(* CODESYS project Box_Sorting.project

Project tree, tasks and I/O mapping:
  Device : CODESYS Control Win V3 x64, 3S - Smart Software Solutions GmbH, version 3.5.16.40
    application Application
      libraries: Standard, * (System)
      task MainTask (cyclic, interval t#20ms, priority 1) calls MainControl
      global variables IOs
      global variables GVL
      Symbols
      visualisation Visualization
      program MainControl [ST]
      program LampCtrl [ST]
      program MainLogic [ST]
      program AlarmHandling [ST]
      program BoxMeasureLogic [ST]
      program SmallBoxLogic [ST]
      program MediumBoxLogic [ST]
      program LargeBoxLogic [ST]
      program AlarmHandlingSUB010 [ST]
      program AlarmHandlingSUB020 [ST]
      program AlarmHandlingSUB030 [ST]
      program AlarmHandlingSUB040 [ST]
      program AlarmHandlingSUB050 [ST]
      program AlarmHandlingCylinder030 [ST]
      program AlarmHandlingCylinder040 [ST]
      program AlarmHandlingCylinder050 [ST]
      program AlarmReset [ST]
  libraries: VisuSymbols, 3.5.10.0 (System)
  text list GlobalTextList
*)

// Device/Application/IOs
VAR_GLOBAL
	//Input
	iSUB010_B1 : BOOL; //Box in position
	iSUB010_B2 : BOOL; //Measure sensor 1, small box
	iSUB010_B3 : BOOL; //Measure sensor 2, medium box
	iSUB010_B4 : BOOL; //Measure sensor 3, large box
	iSUB020_B1 : BOOL; //Small box in position cylinder
	iSUB020_B2 : BOOL; //Medium box in position cylinder
	iSUB020_B3 : BOOL; //Large box in position cylinder
	iSUB030_B1 : BOOL; //Small box first sensor
	iSUB030_B2 : BOOL; //Small box second sensor
	iSUB040_B1 : BOOL; //Medium box first sensor
	iSUB040_B2 : BOOL; //Medium box second sensor
	iSUB050_B1 : BOOL; //Large box first sensor
	iSUB050_B2 : BOOL; //Large box second sensor
	iSUB030_C1_B1 : BOOL; //Small box cylinder max out
	iSUB040_C1_B1 : BOOL; //Medium box cylinder max out
	iSUB050_C1_B1 : BOOL; //Large box cylinder max out
	
	//Output
	oSUB000_H4 : BOOL; //Green light
	oSUB000_H5 : BOOL; //Amber light
	oSUB000_H6 : BOOL; //Red light
	oSUB010_K1 : BOOL; //Sort conveyor
	oSUB020_K1 : BOOL; //Transport conveyor
	oSUB030_K1 : BOOL; //Small box conveyor
	oSUB040_K1 : BOOL; //Medium box conveyor
	oSUB050_K1 : BOOL; //Large box conveyor
	oSUB030_Y1 : BOOL; //Small box cylinder
	oSUB040_Y1 : BOOL; //Medium box cylinder
	oSUB050_Y1 : BOOL; //Large box cylinder

END_VAR

// Device/Application/GVL
VAR_GLOBAL
	
	(*HMI INPUTS*)
	iSUB000_S1: BOOL; 	// Start button
	iSUB000_S2: BOOL := TRUE;  	// Stop button (NC)
	iSUB000_S3: BOOL;	// Reset button

	(*HMI OUTPUTS*)
	oSUB000_H1: BOOL; 	// Start button lamp
	oSUB000_H2: INT; 	// Display
	oSUB000_H3: BOOL; 	// Reset button lamp

END_VAR

// Device/Application/MainControl
PROGRAM MainControl
VAR_INPUT
    iStart : BOOL;   // Start
    iStop  : BOOL;   // Stop
    iFault : BOOL;   // Fault
END_VAR

VAR_OUTPUT
    oRun         : BOOL;   // State Run
    oIdle        : BOOL;   // State Idle
    oFaultActive : BOOL;   // State Faulty
END_VAR

VAR
    Mode : INT := 0;  // 0=Idle, 1=Run, 2=Fault
	prevSUB010_K1 : BOOL;
	prevSUB020_K1 : BOOL;
	prevSUB030_K1 : BOOL;
	prevSUB040_K1 : BOOL;
	prevSUB050_K1 : BOOL;
	valueSaved :BOOL;
	backupSUB010_K1 : BOOL;
	backupSUB020_K1 : BOOL;
	backupSUB030_K1 : BOOL;
	backupSUB040_K1 : BOOL;
	backupSUB050_K1 : BOOL;

	//boxInTransport : BOOL; //a box are deployed and are in transit
END_VAR

AlarmHandling();
iFault := AlarmHandling.alarmActive;

// Huvudlogik
CASE Mode OF
    0: // Idle
        oRun := FALSE;
        oIdle := TRUE;
        oFaultActive := FALSE;
		
		//Save outputs when enter Idle
		IF NOT valueSaved AND NOT iFault THEN
			backupSUB010_K1 := IOs.oSUB010_K1;
			backupSUB020_K1 := IOs.oSUB020_K1;
			backupSUB030_K1 := IOs.oSUB030_K1;
			backupSUB040_K1 := IOs.oSUB040_K1;
			backupSUB050_K1 := IOs.oSUB050_K1;
			valueSaved := TRUE;
		END_IF
        
        IF GVL.iSUB000_S1 THEN //Start
			iStop := FALSE;
			iStart := TRUE;
			IF NOT iFault THEN
            	Mode := 1; // Automatic operation
        	ELSE
            	Mode := 2; //Faulted
			END_IF;
        END_IF;
		
		//Stop output in Idle
		IOs.oSUB010_K1 := FALSE;
		IOs.oSUB020_K1 := FALSE;
		IOs.oSUB030_K1 := FALSE;
		IOs.oSUB040_K1 := FALSE;
		IOs.oSUB050_K1 := FALSE;
		
    1: // Run (Automatic)
        oRun := TRUE;
        oIdle := FALSE;
        oFaultActive := FALSE;
        
		//Restore backup for outputs when we start
		IF valueSaved THEN
			IOs.oSUB010_K1 := backupSUB010_K1;
			IOs.oSUB020_K1 := backupSUB020_K1;
			IOs.oSUB030_K1 := backupSUB030_K1;
			IOs.oSUB040_K1 := backupSUB040_K1;
			IOs.oSUB050_K1 := backupSUB050_K1;
			valueSaved := FALSE;
		END_IF
		
		//Enter Faulty if alarm active
		IF iFault THEN
			//Save all output when alarm
			IF NOT valueSaved THEN
				backupSUB010_K1 := IOs.oSUB010_K1;
				backupSUB020_K1 := IOs.oSUB020_K1;
				backupSUB030_K1 := IOs.oSUB030_K1;
				backupSUB040_K1 := IOs.oSUB040_K1;
				backupSUB050_K1 := IOs.oSUB050_K1;
				valueSaved := TRUE;
			END_IF;
			//Stop output when fault
			IOs.oSUB010_K1 := FALSE;
			IOs.oSUB020_K1 := FALSE;
			IOs.oSUB030_K1 := FALSE;
			IOs.oSUB040_K1 := FALSE;
			IOs.oSUB050_K1 := FALSE;
			
			Mode := 2; //Faulted
		ELSIF NOT GVL.iSUB000_S2 THEN
			iStop := TRUE;
			iStart := FALSE;
			Mode := 0; // Set Idle mode
		ELSE
			MainLogic();
		END_IF
        

    2: // Faulted
        oRun := FALSE;
        oIdle := FALSE;
        oFaultActive := TRUE;
		
		//Stop output when fault
		IOs.oSUB010_K1 := FALSE;
		IOs.oSUB020_K1 := FALSE;
		IOs.oSUB030_K1 := FALSE;
		IOs.oSUB040_K1 := FALSE;
		IOs.oSUB050_K1 := FALSE;
		
		IF GVL.iSUB000_S3 THEN
			iStop := TRUE;
			iStart := FALSE;
			AlarmReset();
			IF NOT IOs.iSUB010_B1 THEN // Prevent alarm 9 to heal if before second box is removed from system
				Mode := 0; // Return to idle
			ELSE //Still keep alarm 9
				AlarmHandling.alarmActive := TRUE;
				AlarmHandling.alarmCode := 9;	
			END_IF
        END_IF;

    ELSE
        Mode := 0; // Failsafe
END_CASE;

//Call lamp control
LampCtrl();

END_PROGRAM

// Device/Application/AlarmHandling
PROGRAM AlarmHandling
VAR_INPUT
	boxInSystem : BOOL; //Box introduced in the system
	alarmActive : BOOL; //If any alarm is active
	alarmCode : INT;  //Alarm code
END_VAR
VAR
END_VAR

//Stop all timers if a alarm is active
IF alarmCode <> 0 THEN
	AlarmHandlingSUB010.startTimeSUB010 := FALSE;
	AlarmHandlingSUB020.startTimeSUB020 := FALSE;
	AlarmHandlingSUB030.startTimeSUB030 := FALSE;
	AlarmHandlingSUB040.startTimeSUB040 := FALSE;
	AlarmHandlingSUB050.startTimeSUB050 := FALSE;
	AlarmHandlingCylinder030.startTimeCyl030 := FALSE;
	AlarmHandlingCylinder040.startTimeCyl040 := FALSE;
	AlarmHandlingCylinder050.startTimeCyl050 := FALSE;
END_IF
AlarmHandlingSUB010();
AlarmHandlingSUB020();
AlarmHandlingSUB030();
AlarmHandlingSUB040();
AlarmHandlingSUB050();
AlarmHandlingCylinder030();
AlarmHandlingCylinder040();
AlarmHandlingCylinder050();

//Display the Alarm code
oSUB000_H2 := alarmCode;

END_PROGRAM

// Device/Application/AlarmHandlingSUB010
PROGRAM AlarmHandlingSUB010
VAR_INPUT
	startTimeSUB010 : BOOL; //Activate timer
	SUB010Timer : TON;  //Alarm timer
END_VAR
VAR
	boxStart : F_TRIG; // Instance of flankdetector, control when box is on the conveyour
END_VAR

//Alarmhandling Conveyour 1, SUB010
boxStart(CLK := IOs.iSUB010_B1);
IF boxStart.Q THEN
	AlarmHandling.boxInSystem := TRUE;
	startTimeSUB010 := TRUE;
ELSIF IOs.iSUB010_B1 AND AlarmHandling.boxInSystem AND NOT MainControl.iStop THEN
	AlarmHandling.alarmActive := TRUE;
	IF AlarmHandling.alarmCode = 0 THEN
		AlarmHandling.alarmCode := 9;
	END_IF;
END_IF
IF IOs.iSUB010_B2 OR MainControl.iStop THEN //Cancel alarm
	startTimeSUB010 := FALSE;
END_IF
IF SUB010Timer.Q AND (AlarmHandling.alarmCode = 0) THEN
	AlarmHandling.alarmActive := TRUE;
	AlarmHandling.alarmCode := 1;
END_IF
SUB010Timer(IN := startTimeSUB010, PT := T#4S);

END_PROGRAM

// Device/Application/AlarmHandlingSUB020
PROGRAM AlarmHandlingSUB020
VAR_INPUT
	startTimeSUB020 : BOOL; //Activate timer
	SUB020Timer : TON;  //Alarm timer
END_VAR
VAR
END_VAR

//Alarmhandling Conveyour 2, SUB020
IF IOs.iSUB010_B2 AND (AlarmHandling.alarmCode = 0) AND NOT MainControl.iStop THEN
	startTimeSUB020 := TRUE;
END_IF
IF IOs.iSUB020_B1 AND (MainLogic.boxSize = 1) THEN //Cancel alarm when reach small box sensor, small box
	startTimeSUB020 := FALSE;
ELSIF IOs.iSUB020_B2 AND (MainLogic.boxSize = 2) THEN //Cancel alarm when reach medium box sensor, medium box
	startTimeSUB020 := FALSE;
ELSIF IOs.iSUB020_B3 AND (MainLogic.boxSize = 3) THEN //Cancel alarm when reach large box sensor, large box
	startTimeSUB020 := FALSE;
ELSIF MainControl.iStop THEN
	startTimeSUB020 := FALSE;
END_IF
IF SUB020Timer.Q AND (AlarmHandling.alarmCode = 0) THEN
	AlarmHandling.alarmActive := TRUE;
	AlarmHandling.alarmCode := 2;
END_IF
SUB020Timer(IN := startTimeSUB020, PT := T#8S);

END_PROGRAM

// Device/Application/MainLogic
PROGRAM MainLogic
VAR_INPUT
	boxSize : INT; //Size of the Box
END_VAR
VAR
END_VAR

IF boxSize = 0 THEN  //Box to measure
	BoxMeasureLogic();
ELSIF boxSize = 1 THEN //Small box
	SmallBoxLogic();
ELSIF BoxSize = 2 THEN //Medium box
	MediumBoxLogic();
ELSIF boxSize = 3 THEN //Large box
	LargeBoxLogic();
END_IF

END_PROGRAM

// Device/Application/BoxMeasureLogic
PROGRAM BoxMeasureLogic
VAR
END_VAR

//Start conveyor 1
IF MainControl.oRun AND IOs.iSUB010_B1 THEN
	IOs.oSUB010_K1 := TRUE;
END_IF
//Measure Box size, Small =1, Medium =2, Large =3.
IF IOs.iSUB010_B2 THEN
	MainLogic.boxSize := 1;
	IF IOs.iSUB010_B3 THEN
		MainLogic.boxSize := 2;
		IF IOs.iSUB010_B4 THEN
			MainLogic.boxSize := 3;
		END_IF
	END_IF
END_IF
//Start conveyor 2
IF MainLogic.boxSize > 0 AND IOs.oSUB010_K1 THEN
	IOs.oSUB020_K1 := TRUE;
END_IF

END_PROGRAM

// Device/Application/SmallBoxLogic
PROGRAM SmallBoxLogic
VAR
END_VAR

//Check if Box size is small at cylinder_small. If small Box, stop conveyor and push Box to conveyor 3
IF IOs.iSUB020_B1 THEN
	IOs.oSUB010_K1 := FALSE; //Stop conveyor 1
	IF MainLogic.boxSize = 1 THEN
		IOs.oSUB020_K1 := FALSE; //Stop conveyor 2
		IOs.oSUB030_Y1 := TRUE;  //Expand cylinder small
	END_IF
END_IF

//When cylinder small is fully out and first sensor on conveyor 3 is akitve, start conveyor 3
IF IOs.iSUB030_C1_B1 AND IOs.iSUB030_B1 THEN
	IOs.oSUB030_Y1 := FALSE;  //Retract cylinder small
	IOs.oSUB030_K1 := TRUE;
END_IF

//Stop conveyor 3 when it reach second sensor
IF IOs.iSUB030_B2 THEN
	IOs.oSUB030_K1 := FALSE;
	MainLogic.boxSize := 0;
END_IF

END_PROGRAM

// Device/Application/MediumBoxLogic
PROGRAM MediumBoxLogic
VAR
END_VAR

//Check if Box size is medium at cylinder_medium. If medium Box, stop conveyor and push Box to conveyor 4
IF MainLogic.boxSize = 2 AND IOs.iSUB020_B2 THEN
	IOs.oSUB010_K1 := FALSE; //Stop conveyor 1
	IOs.oSUB020_K1 := FALSE; //Stop conveyor 2
	IOs.oSUB040_Y1 := TRUE;  //Expand cylinder medium
END_IF

//When cylinder medium is fully out and first sensor on conveyor 4 is akitve, start conveyor 4
IF IOs.iSUB040_C1_B1 AND IOs.iSUB040_B1 THEN
	IOs.oSUB040_Y1 := FALSE;  //Retract cylinder medium
	IOs.oSUB040_K1 := TRUE; //Start conveyor 4
END_IF

//Stop conveyor 4 when it reach second sensor
IF IOs.iSUB040_B2 THEN
	IOs.oSUB040_K1 := FALSE;
	MainLogic.boxSize := 0;
END_IF

END_PROGRAM

// Device/Application/LargeBoxLogic
PROGRAM LargeBoxLogic
VAR
END_VAR

//Check if Box size is large at cylinder_large. If large Box, stop conveyor and push Box to conveyor 5
IF MainLogic.boxSize = 3 AND IOs.iSUB020_B3 THEN
	IOs.oSUB010_K1 := FALSE; //Stop conveyor 1
	IOs.oSUB020_K1 := FALSE; //Stop conveyor 2
	IOs.oSUB050_Y1 := TRUE;  //Expand cylinder large
END_IF

//When cylinder large is fully out and first sensor on conveyor 5 is aktive, start conveyor 5
IF IOs.iSUB050_C1_B1 AND IOs.iSUB050_B1 THEN
	IOs.oSUB050_Y1 := FALSE;  //Retract cylinder large
	IOs.oSUB050_K1 := TRUE; //Start conveyor 5
END_IF

//Stop conveyor 5 when it reach second sensor
IF IOs.iSUB050_B2 THEN
	IOs.oSUB050_K1 := FALSE;
	MainLogic.boxSize := 0;
END_IF

END_PROGRAM

// Device/Application/AlarmHandlingSUB030
PROGRAM AlarmHandlingSUB030
VAR_INPUT
	startTimeSUB030 : BOOL; //Activate timer
	SUB030Timer : TON; //Alarm timer
END_VAR
VAR
	boxEndSmall : F_TRIG; // Instance of flankdetector, control when box is removed
END_VAR

//Alarmhandling Conveyour 3, SUB030
IF IOs.iSUB030_B1 AND (AlarmHandling.alarmCode = 0) AND NOT MainControl.iStop THEN
	startTimeSUB030 := TRUE;
END_IF
boxEndSmall(CLK := IOs.iSUB030_B2);
IF boxEndSmall.Q THEN //Cancel alarm
	startTimeSUB030 := FALSE;
	IF NOT IOs.iSUB030_B2 THEN
		AlarmHandling.boxInSystem := FALSE;
	END_IF
ELSIF MainControl.iStop THEN
	startTimeSUB030 := FALSE;
END_IF
IF SUB030Timer.Q AND (AlarmHandling.alarmCode = 0) THEN
	AlarmHandling.alarmActive := TRUE;
	AlarmHandling.alarmCode := 3;
END_IF
SUB030Timer(IN := startTimeSUB030, PT := T#7.2S);

END_PROGRAM

// Device/Application/AlarmHandlingSUB040
PROGRAM AlarmHandlingSUB040
VAR_INPUT
	startTimeSUB040 : BOOL; //Activate timer
	SUB040Timer : TON;  //Alarm timer
END_VAR
VAR
	boxEndMedium : F_TRIG; // Instance of flankdetector, control when box is removed
END_VAR

//Alarmhandling Conveyour 4, SUB040
IF IOs.iSUB040_B1 AND (AlarmHandling.alarmCode = 0) AND NOT MainControl.iStop THEN
	startTimeSUB040 := TRUE;
END_IF
boxEndMedium(CLK := IOs.iSUB040_B2);
IF boxEndMedium.Q THEN //Cancel alarm
	startTimeSUB040 := FALSE;
	IF NOT IOs.iSUB040_B2 THEN
		AlarmHandling.boxInSystem := FALSE;
	END_IF
ELSIF MainControl.iStop THEN
	startTimeSUB040 := FALSE;
END_IF
IF SUB040Timer.Q AND (AlarmHandling.alarmCode = 0) THEN
	AlarmHandling.alarmActive := TRUE;
	AlarmHandling.alarmCode := 4;
END_IF
SUB040Timer(IN := startTimeSUB040, PT := T#7.3S);

END_PROGRAM

// Device/Application/AlarmHandlingSUB050
PROGRAM AlarmHandlingSUB050
VAR_INPUT
	startTimeSUB050 : BOOL; //Activate timer
	SUB050Timer : TON;  //Alarm timer
END_VAR
VAR
	boxEndLarge : F_TRIG; // Instance of flankdetector, control when box is removed
END_VAR

//Alarmhandling Conveyour 5, SUB050
IF IOs.iSUB050_B1 AND (AlarmHandling.alarmCode = 0) AND NOT MainControl.iStop THEN
	startTimeSUB050 := TRUE;
END_IF
boxEndLarge(CLK := IOs.iSUB050_B2);
IF boxEndLarge.Q THEN //Cancel alarm
	startTimeSUB050 := FALSE;
	IF NOT IOs.iSUB050_B2 THEN
		AlarmHandling.boxInSystem := FALSE;
	END_IF
ELSIF MainControl.iStop THEN
	startTimeSUB050 := FALSE;
END_IF
IF SUB050Timer.Q AND (AlarmHandling.alarmCode = 0) THEN
	AlarmHandling.alarmActive := TRUE;
	AlarmHandling.alarmCode := 5;
END_IF
SUB050Timer(IN := startTimeSUB050, PT := T#7.4S);

END_PROGRAM

// Device/Application/AlarmHandlingCylinder030
PROGRAM AlarmHandlingCylinder030
VAR_INPUT
	Cyl030Timer : TON; //Alarm timer
	startTimeCyl030 : BOOL; //Activate timer
END_VAR
VAR
END_VAR

//Alarmhandling Cylinder small, SUB030Cylinder
//Cylinder do not expand
IF IOs.iSUB020_B1 AND (MainLogic.boxSize = 1) AND NOT MainControl.iStop THEN
	startTimeCyl030 := TRUE;
END_IF
IF IOs.iSUB030_B1 THEN //Cancel alarm
	startTimeCyl030 := FALSE;
END_IF
IF Cyl030Timer.Q AND (AlarmHandling.alarmCode = 0) THEN
	AlarmHandling.alarmActive := TRUE;
	AlarmHandling.alarmCode := 6;
END_IF
Cyl030Timer(IN := startTimeCyl030, PT := T#6.5S);

END_PROGRAM

// Device/Application/AlarmHandlingCylinder040
PROGRAM AlarmHandlingCylinder040
VAR_INPUT
	Cyl040Timer : TON; //Alarm timer
	startTimeCyl040 : BOOL; //Activate timer
END_VAR
VAR
END_VAR

//Alarmhandling Cylinder medium, SUB040Cylinder
//Cylinder do not expand
IF IOs.iSUB020_B2 AND (MainLogic.boxSize = 2) AND NOT MainControl.iStop THEN
	startTimeCyl040 := TRUE;
END_IF
IF IOs.iSUB040_B1 THEN //Cancel alarm
	startTimeCyl040 := FALSE;
END_IF
IF Cyl040Timer.Q AND (AlarmHandling.alarmCode = 0) THEN
	AlarmHandling.alarmActive := TRUE;
	AlarmHandling.alarmCode := 7;
END_IF
Cyl040Timer(IN := startTimeCyl040, PT := T#6.6S);

END_PROGRAM

// Device/Application/AlarmHandlingCylinder050
PROGRAM AlarmHandlingCylinder050
VAR_INPUT
	Cyl050Timer : TON; //Alarm timer
	startTimeCyl050 : BOOL; //Activate timer
END_VAR
VAR
END_VAR

//Alarmhandling Cylinder large, SUB050Cylinder
//Cylinder do not expand
IF IOs.iSUB020_B3 AND (MainLogic.boxSize = 3) AND NOT MainControl.iStop THEN
	startTimeCyl050 := TRUE;
END_IF
IF IOs.iSUB050_B1 THEN //Cancel alarm
	startTimeCyl050 := FALSE;
END_IF
IF Cyl050Timer.Q AND (AlarmHandling.alarmCode = 0) THEN
	AlarmHandling.alarmActive := TRUE;
	AlarmHandling.alarmCode := 8;
END_IF
Cyl050Timer(IN := startTimeCyl050, PT := T#6.7S);

END_PROGRAM

// Device/Application/AlarmReset
PROGRAM AlarmReset
VAR
END_VAR

//Reset alarm
AlarmHandling.alarmActive := FALSE;
AlarmHandlingSUB010.startTimeSUB010 := FALSE;
AlarmHandlingSUB020.startTimeSUB020 := FALSE;
AlarmHandlingSUB030.startTimeSUB030 := FALSE;
AlarmHandlingSUB040.startTimeSUB040 := FALSE;
AlarmHandlingSUB050.startTimeSUB050 := FALSE;
AlarmHandlingSUB010.SUB010Timer(IN := AlarmHandlingSUB010.startTimeSUB010);
AlarmHandlingSUB020.SUB020Timer(IN := AlarmHandlingSUB020.startTimeSUB020);
AlarmHandlingSUB030.SUB030Timer(IN := AlarmHandlingSUB030.startTimeSUB030);
AlarmHandlingSUB040.SUB040Timer(IN := AlarmHandlingSUB040.startTimeSUB040);
AlarmHandlingSUB050.SUB050Timer(IN := AlarmHandlingSUB050.startTimeSUB050);
AlarmHandlingCylinder030.startTimeCyl030 := FALSE;
AlarmHandlingCylinder040.startTimeCyl040 := FALSE;
AlarmHandlingCylinder050.startTimeCyl050 := FALSE;
AlarmHandlingCylinder030.Cyl030Timer(IN := AlarmHandlingCylinder030.startTimeCyl030);
AlarmHandlingCylinder040.Cyl040Timer(IN := AlarmHandlingCylinder040.startTimeCyl040);
AlarmHandlingCylinder050.Cyl050Timer(IN := AlarmHandlingCylinder050.startTimeCyl050);
AlarmHandling.alarmCode := 0;

END_PROGRAM

// Device/Application/LampCtrl
PROGRAM LampCtrl
VAR
	GreenBlink : TON; //Green light blink timer
	RedBlink : TON;   //Red light blink timer 
END_VAR

IF MainControl.oRun THEN
	IOs.oSUB000_H4 := TRUE;
	IOs.oSUB000_H5 := FALSE;
	IOs.oSUB000_H6 := FALSE;
	oSUB000_H1 := TRUE;
	oSUB000_H3 := FALSE;
ELSIF MainControl.oIdle THEN
	IOs.oSUB000_H4 := FALSE;
	IOs.oSUB000_H5 := TRUE;
	IOs.oSUB000_H6 := FALSE;
	GreenBlink(IN := NOT GreenBlink.Q, PT := T#2S);
	oSUB000_H1 := GreenBlink.ET > T#1S; //Green shall blink in IDLE
	oSUB000_H3 := FALSE;
ELSIF MainControl.oFaultActive THEN
	IOs.oSUB000_H4 := FALSE;
	IOs.oSUB000_H5 := FALSE;
	oSUB000_H1 := FALSE;
	RedBlink(IN := NOT RedBlink.Q, PT := T#2S);
	IOs.oSUB000_H6 := oSUB000_H3 := RedBlink.ET > T#1S; //Red shall blink in Faulty
END_IF

END_PROGRAM

// Device/Application/Visualization
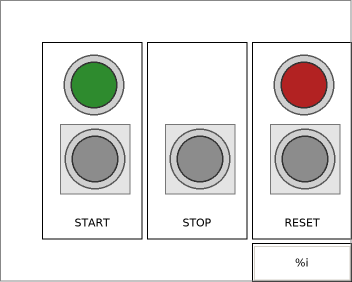
VISUALIZATION Visualization  // 352x282
    Rectangle (42,42 100x197)
    Lamp1 (59,50 70x70), variable: oSUB000_H1, style: Lamp-Lamp1-Green
    PushSwitch (60,124 70x70), variable: iSUB000_S1, behaviour: TAP, style: Switch-PushSwitch-Gray
    Label (46,208 92x30), "START"
    Rectangle (147,42 100x197)
    PushSwitch (165,124 70x70), variable: iSUB000_S2, behaviour: TAP, style: Switch-PushSwitch-Gray
    Label (151,208 92x30), "STOP"
    Rectangle (252,42 100x197)
    Lamp1 (269,50 70x70), variable: oSUB000_H3, style: Lamp-Lamp1-Red
    PushSwitch (270,124 70x70), variable: iSUB000_S3, behaviour: TAP, style: Switch-PushSwitch-Gray
    Label (256,208 92x30), "RESET"
    Rectangle (252,243 100x39)
    Textfield (254,246 96x34), "%i", text variable: oSUB000_H2
END_VISUALIZATION
